FUNCTION_BLOCK CoE_property_usint EXTENDS CoE_property
VAR_INPUT
END_VAR
VAR_OUTPUT
END_VAR
VAR
	_value : USINT;
END_VAR

SUPER^();

PROPERTY dataTypeSize : UINT
GET
dataTypeSize := SIZEOF(_value);
END_GET
END_PROPERTY

METHOD get_value : BOOL
VAR_OUTPUT
	value : usINT ;
	errId : UDINT;
END_VAR
IF init_done THEN
	value := _value;
	get_value := TRUE;
ELSE
	errId := 2;
	get_value := FALSE;
END_IF
END_METHOD

METHOD handle_read_callback : BOOL
VAR_INPUT
	pt_buffer : POINTER TO CoE_buffer_type_cast_union;
	errId : UDINT;
END_VAR

_value := pt_buffer^.value_usint;
_init_done:=TRUE;
_read_errId:=errId;
END_METHOD

METHOD set_value : BOOL
VAR_INPUT
	value : USINT ;
END_VAR
_valueToWrite.value_usint := value;
IF THIS^._CoE_property_handler <> 0 THEN 
	THIS^._CoE_property_handler.add_write_request(THIS^);
ELSE
	errId:=1;
END_IF
END_METHOD

END_FUNCTION_BLOCK

(* stored: Version 1.1.0.1, ProductVersion 3.1.4024.6
   POU CoE_property_usint: Id {0f249b99-a993-089f-0673-1d159a29be72}, SpecialFunc None
   Property dataTypeSize: Id {91f35848-1c7b-078a-0496-e0009e5a7dee}
   Get Get: Id {643eca5b-2bf9-0a60-2d7a-471a753c2851}
   Method get_value: Id {59517984-c58f-0bc2-19c4-bd11556a6453}
   Method handle_read_callback: Id {23eac60e-5a02-02cf-18d0-a28bcb92ebe7}
   Method set_value: Id {64aa3150-9efa-04f2-22f9-861eadf4c280} *)
